FUNCTION_BLOCK ASRT_AX_T_FF_SR (* Event-driven bistable and Toggle *)
  (* Standard: 61499-1 Annex A; Description: Copyright (c) 2026 HR Agrartechnik GmbH This program and the accompanying materials are made available under the terms of the Eclipse Public License 2.0 which is available at https://www.eclipse.org/legal/epl-2.0/ SPDX-License-Identifier: EPL-2.0 *)
  (* Version 1.0, 2026-09-03, Franz Höpfinger, HR Agrartechnik GmbH, wie ASR_AX_SR, aber fuer AX_T_FF_SR (S/R/CLK als ASRT-Socket statt 3 einzelner EventInputs) *)
  PACKAGE adapter::events::unidirectional;
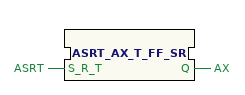
  SOCKETS
    S_R_T : adapter::types::unidirectional::ASRT; (* Set/Reset/Toggle *)
  END_SOCKETS
  PLUGS
    Q : adapter::types::unidirectional::AX; (* value of flip flop *)
  END_PLUGS
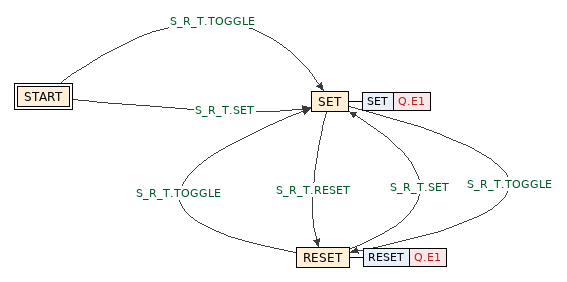
  EC_STATES
    START; (* Initial State *)
    SET : SET -> Q.E1;
    RESET : RESET -> Q.E1;
  END_STATES
  EC_TRANSITIONS
    START TO SET := S_R_T.SET;
    SET TO RESET := S_R_T.RESET;
    RESET TO SET := S_R_T.SET;
    SET TO RESET := S_R_T.TOGGLE;
    RESET TO SET := S_R_T.TOGGLE;
    START TO SET := S_R_T.TOGGLE;
  END_TRANSITIONS
  ALGORITHM SET IN ST:
Q.D1 := TRUE;
  END_ALGORITHM
  ALGORITHM RESET IN ST:
Q.D1 := FALSE;
  END_ALGORITHM
END_FUNCTION_BLOCK
